  kill rq_gripper_communication_thread
  rq_gripper_communication_thread_started = False
  rq_close_gripper_socket("1")
  rq_close_gripper_socket("2")
  rq_close_gripper_socket("3")
  rq_close_gripper_socket("4")

  rq_init_comm_if_connected(9, "1")
  rq_init_comm_if_connected(2, "2")
  rq_init_comm_if_connected(3, "3")
  rq_init_comm_if_connected(4, "4")
  rq_print_connected_grippers()
  rq_gripper_communication_thread = run rq_gripper_communication()

  while(not rq_gripper_communication_thread_started):
      sleep(0.008)
  end

  rq_set_max_current_for_all_grippers()

  reset_and_activate = False

  rq_activate_all_grippers(False)
  # end: URCap Program Node
  # begin: URCap Program Node
  #   Source: Robotiq_Grippers, 1.8.9.14887, Robotiq Inc.
  #   Type: Gripper
  $ 52 "Gripper Move70% (1)"
  if not(gripper_connected[0]):
    popup("Gripper 1 must be connected to run this program.", "No connection", False, True, True)
  end
  if not(rq_is_gripper_activated("1")):
    popup("Gripper 1 is not activated. Go to Installation tab > Gripper to activate it and run the program again.", "Not activated", False, True, True)
  end
  rq_set_pos_spd_for(179, 255, 0, "1")
  rq_wait_pos_spe_for_request(179, 255, 0, "1")
  rq_go_to("1")
  rq_wait("1")
  # end: URCap Program Node
  $ 53 "Waypoint_31" "breakAfter"
  movej(get_inverse_kin(Waypoint_31_p, qnear=Waypoint_31_q), a=1.3962634015954636, v=1.0471975511965976)
  $ 54 "Waypoint_27" "breakAfter"
  movej(get_inverse_kin(Waypoint_27_p, qnear=Waypoint_27_q), a=1.3962634015954636, v=1.0471975511965976)
  $ 55 "stick1" "breakAfter"
  movej(get_inverse_kin(stick1_p, qnear=stick1_q), a=1.3962634015954636, v=1.0471975511965976)
  # begin: URCap Program Node
  #   Source: Robotiq_Grippers, 1.8.9.14887, Robotiq Inc.
  #   Type: Gripper
  $ 56 "Gripper Close (1)"
  if not(gripper_connected[0]):
    popup("Gripper 1 must be connected to run this program.", "No connection", False, True, True)
  end
  if not(rq_is_gripper_activated("1")):
    popup("Gripper 1 is not activated. Go to Installation tab > Gripper to activate it and run the program again.", "Not activated", False, True, True)
  end
  rq_set_pos_spd_for(255, 0, 0, "1")
  rq_wait_pos_spe_for_request(255, 0, 0, "1")
  rq_go_to("1")
  rq_wait("1")
  # end: URCap Program Node
  $ 57 "Waypoint_3" "breakAfter"
  movej(get_inverse_kin(Waypoint_3_p, qnear=Waypoint_3_q), a=1.3962634015954636, v=1.0471975511965976)
  $ 58 "Waypoint_4" "breakAfter"
  movej(get_inverse_kin(Waypoint_4_p, qnear=Waypoint_4_q), a=1.3962634015954636, v=1.0471975511965976)
  $ 59 "Waypoint_30" "breakAfter"
  movej(get_inverse_kin(Waypoint_30_p, qnear=Waypoint_30_q), a=1.3962634015954636, v=1.0471975511965976)
  $ 60 "Waypoint_28" "breakAfter"
  movej(get_inverse_kin(Waypoint_28_p, qnear=Waypoint_28_q), a=1.3962634015954636, v=1.0471975511965976)
  $ 61 "Waypoint_24" "breakAfter"
  movej(get_inverse_kin(Waypoint_24_p, qnear=Waypoint_24_q), a=1.3962634015954636, v=1.0471975511965976)
  $ 62 "Waypoint_23" "breakAfter"
  movej(get_inverse_kin(Waypoint_23_p, qnear=Waypoint_23_q), a=1.3962634015954636, v=1.0471975511965976)
  $ 63 "center1" "breakAfter"
  movej(get_inverse_kin(center1_p, qnear=center1_q), a=1.3962634015954636, v=1.0471975511965976)
  $ 64 "'Now Cotton Candy Creation'"
  # 'Now Cotton Candy Creation'
  $ 66 "radius≔0.13"
  global radius=0.13
  $ 67 "height≔0.05"
  global height=0.05
  $ 72 "start_wait≔1"
  global start_wait=1
  $ 73 "start_time≔33.75"
  global start_time=33.75
  $ 74 "circle_time≔3.75"
  global circle_time=3.75
  $ 77 "center≔Tool_const"
  global center=get_forward_kin()
  $ 78 "bottom≔pose_add(center, p[0, -radius, height, 0, 0, 0])"
  global bottom= pose_add (center, p[0, -radius, height, 0, 0, 0])
  $ 79 "right≔pose_add(center, p[-radius, 0, -height, 0, 0, 0])"
  global right= pose_add (center, p[-radius, 0, -height, 0, 0, 0])
  $ 80 "top_circ≔pose_add(center, p[0, radius, height, 0, 0, 0])"
  global top_circ= pose_add (center, p[0, radius, height, 0, 0, 0])
  $ 81 "left≔pose_add(center, p[radius, 0, -height, 0, 0, 0])"
  global left= pose_add (center, p[radius, 0, -height, 0, 0, 0])
  $ 95 "timer_3: Stop"
  timer_3_is_counting = False
  $ 98 "sleep(start_wait)"
  sleep(start_wait)
  $ 99 "timer_1: Start"
  timer_1_is_counting = True
  $ 100 "Loop start_time>0"
  while (start_time>0):
    $ 101 "MoveP"
    $ 102 "bottom" "breakAfter"
    movep(bottom, a=1.2, v=0.25, r=0.125)
    $ 103 "CircleMove"
    $ 104 "left" "noBreak"
    $ 105 "top_circ" "breakAfter"
    movec(left, top_circ, a=1.2, v=0.25, r=0.125)
    $ 106 "MoveP"
    $ 107 "top_circ" "breakAfter"
    movep(top_circ, a=1.2, v=0.25, r=0.025)
    $ 108 "CircleMove"
    $ 109 "right" "noBreak"
    $ 110 "bottom" "breakAfter"
    movec(right, bottom, a=1.2, v=0.25, r=0.025)
    $ 115 "start_time≔start_time-circle_time"
    global start_time=start_time-circle_time
  end
  $ 116 "timer_1: Stop"
  timer_1_is_counting = False
  $ 117 "MoveL"
  $ 118 "Waypoint_2" "breakAfter"
  movel(Waypoint_2_p, a=1.2, v=0.25)
  $ 119 "Waypoint_5" "breakAfter"
  movel(Waypoint_5_p, a=1.2, v=0.25)
  $ 120 "Waypoint_25" "breakAfter"
  movel(Waypoint_25_p, a=1.2, v=0.25)
  $ 121 "Waypoint_12" "breakAfter"
  movel(Waypoint_12_p, a=1.2, v=0.25)
  $ 122 "Waypoint_13" "breakAfter"
  movel(Waypoint_13_p, a=1.2, v=0.25)
  $ 123 "Waypoint_11" "breakAfter"
  movel(Waypoint_11_p, a=1.2, v=0.25)
  # begin: URCap Program Node
  #   Source: Robotiq_Grippers, 1.8.9.14887, Robotiq Inc.
  #   Type: Gripper Activate
  $ 124 "Gripper Activate"

  kill rq_gripper_communication_thread
  rq_gripper_communication_thread_started = False
  rq_close_gripper_socket("1")
  rq_close_gripper_socket("2")
  rq_close_gripper_socket("3")
  rq_close_gripper_socket("4")

  rq_init_comm_if_connected(9, "1")
  rq_init_comm_if_connected(2, "2")
  rq_init_comm_if_connected(3, "3")
  rq_init_comm_if_connected(4, "4")
  rq_print_connected_grippers()
  rq_gripper_communication_thread = run rq_gripper_communication()

  while(not rq_gripper_communication_thread_started):
      sleep(0.008)
  end

  rq_set_max_current_for_all_grippers()

  reset_and_activate = False

  rq_activate_all_grippers(False)
  # end: URCap Program Node
  # begin: URCap Program Node
  #   Source: Robotiq_Grippers, 1.8.9.14887, Robotiq Inc.
  #   Type: Gripper
  $ 125 "Gripper Open (1)"
  if not(gripper_connected[0]):
    popup("Gripper 1 must be connected to run this program.", "No connection", False, True, True)
  end
  if not(rq_is_gripper_activated("1")):
    popup("Gripper 1 is not activated. Go to Installation tab > Gripper to activate it and run the program again.", "Not activated", False, True, True)
  end
  rq_set_pos_spd_for(0, 255, 0, "1")
  rq_wait_pos_spe_for_request(0, 255, 0, "1")
  rq_go_to("1")
  rq_wait("1")
  # end: URCap Program Node
  $ 126 "Waypoint_14" "breakAfter"
  movel(Waypoint_14_p, a=1.2, v=0.25)
  # begin: URCap Program Node
  #   Source: Robotiq_Grippers, 1.8.9.14887, Robotiq Inc.
  #   Type: Gripper
  $ 127 "Gripper Close (1)"
  if not(gripper_connected[0]):
    popup("Gripper 1 must be connected to run this program.", "No connection", False, True, True)
  end
  if not(rq_is_gripper_activated("1")):
    popup("Gripper 1 is not activated. Go to Installation tab > Gripper to activate it and run the program again.", "Not activated", False, True, True)
  end
  rq_set_pos_spd_for(255, 255, 0, "1")
  rq_wait_pos_spe_for_request(255, 255, 0, "1")
  rq_go_to("1")
  rq_wait("1")
  # end: URCap Program Node
  $ 128 "MoveL"
  $ 129 "Waypoint_15" "breakAfter"
  movel(Waypoint_15_p, a=1.2, v=0.25)
  $ 130 "Waypoint_16" "breakAfter"
  movel(Waypoint_16_p, a=1.2, v=0.25)
  $ 131 "Waypoint_17" "breakAfter"
  movel(Waypoint_17_p, a=1.2, v=0.25)
  $ 132 "Waypoint_6" "breakAfter"
  movel(Waypoint_6_p, a=1.2, v=0.25)
  $ 133 "Waypoint_18" "breakAfter"
  movel(Waypoint_18_p, a=1.2, v=0.25)
  $ 134 "timer_2: Stop"
  timer_2_is_counting = False
  $ 136 "sleep(5)"
  sleep(5)
  $ 137 "Waypoint_20" "breakAfter"
  movel(Waypoint_20_p, a=1.2, v=0.25)
  $ 138 "base_position_2" "breakAfter"
  movel(base_position_2_p, a=1.2, v=0.25)
  $ 139 "Waypoint_22" "breakAfter"
  movel(Waypoint_22_p, a=1.2, v=0.25)
  $ 140 "base_position_1" "breakAfter"
  movel(base_position_1_p, a=1.2, v=0.25)
end
